FUNCTION F_SAFETY_AnzeigenHohePrio : BOOL (* Ehemals F_PNOZ_AnzeigenHohePrio() *)
VAR_INPUT
END_VAR
VAR
END_VAR

(*    
	  U     "T 72"
      SPB   POK
*)
IF GVL.tonSAFETYok.Q THEN //(ehem. T72)
	RETURN;
END_IF


(*
      L     27  //PNOZ-Signal ungültig
      T     "DB6".w226_Betr_Anz_Wert
*)
DB6.w226_Betr_Anz_Wert := 127;

(*
      L     "DB6".w230
      L     24
      ==I   
      SPBN  a01
*)
IF (* DB6.w230 = 24 *) NOT IO.safeOutHauptLuft THEN
	(*
	 L    1                           //Druckluft nicht ein (weiter mit Masch-Ein)
	 T     "DB6".w226_Betr_Anz_Wert
	*)
	DB6.w226_Betr_Anz_Wert := 101;
END_IF
(*	  
a01:  BLD   130
      L     "DB6".w230
      L     48
      ==I   
      SPBN  a02
*)
IF (* DB6.w230 = 48 *) NOT IO.safeOutHauptLuft AND NOT IO.safeOutSchutzTueren THEN
	(*
	L     2   //Schutztür nicht zu
    T     "DB6".w226_Betr_Anz_Wert
	*)
	DB6.w226_Betr_Anz_Wert := 102;
END_IF
(*	  
      
a02:  BLD   130
      L     "DB6".w230
      L     68
      ==I   
      SPBN  a05
*)
IF (* DB6.w230 = 68 *) NOT IO.inResetNotHalt THEN
	(*
	L     5  //Kein Signal von Taste Maschine-Aus
    T     "DB6".w226_Betr_Anz_Wert
	*)
	DB6.w226_Betr_Anz_Wert := 105;
END_IF
(*	  
a05:  BLD   130
      L     "DB6".w230
      L     72
      ==I   
      SPBN  a08
*)
IF (* DB6.w230 = 72 *) NOT IO.safeOutHauptLuft AND NOT IO.safeOutNotHalt THEN
	(*
	 L     8                           //Not-Aus Steuerpult nicht OK     
     T     "DB6".w226_Betr_Anz_Wert
	*)
	DB6.w226_Betr_Anz_Wert := 108;
END_IF




(*	  
a08:  BLD   130
      U     "T 70"
      SPBN  a09
*)


//IF NOT GVL.tonPnozEntprell.Q THEN
//	RETURN;
//END_IF
(*
      L     9                           //Kein Signal von PNOZ
      T     "DB6".w226_Betr_Anz_Wert
*)
//DB6.w226_Betr_Anz_Wert := 109;
(*
a09:  BLD   130
POK:  BLD   130
*)

END_FUNCTION

(* stored: Version 1.1.0.1, ProductVersion 3.1.4024.3
   POU F_SAFETY_AnzeigenHohePrio: Id {003bd5c4-83cf-4cd1-8fbf-5b9eac48c75d}, SpecialFunc None *)
